// TIA Portal V18 export
TYPE "UDT_DLsAI"
// stored: IsFailsafeCompliant false
   STRUCT
      rDayTankLevel : Array[1..2] of Real;   // 10.82(3) Рівень палива в баку добового запасу ДГУ1(2)
   END_STRUCT;
END_TYPE
